PROGRAM ITAction
(*IMPORTANT !!! à modifier correctment selon les besoins*)
VAR CONSTANT
	//nombre total de dynamixel
	iNombreDynamixel 	: INT := 4;
	iNombreXL			: INT := 2;
	iNombreAX			: INT := 2;
	
	//définition de l'ID des dynamixels, tous les ID doivent se suivrent => ex: moteur_1 := 1,moteur_2 := 2, moteur_3 := 3, etc...
	//Si des moteurs AX-12A sont présents, leur ID doivent aller après celles des moteurs XL430 ou XL330 => ex: XL430_moteur_5 := 5, AX12A_moteur_1 := 6, etc...
	MoteurXL1 			: INT := 1; //exemple XL430
	MoteurXL2			: INT := 2;
	MoteurAX1 			: INT := 3; //exemple AX12A
	MoteurAX2			: INT := 4;
END_VAR	

VAR_INPUT
	//démarrage et arrêt du script python
	IbStartPyscript 	: BOOL;
	IbStopPyscript		: BOOL;

	//envoi de commande aux moteurs Dynamixel
	DXLIN 				: ARRAY [1..iNombreDynamixel] OF ST_Dynamixel_Control_Input;
END_VAR

VAR_OUTPUT
	QbPyScriptRunning 	: BOOL; //le script python est actif
	QiNombreDynamixel	: INT;
	//retour d'informations des moteurs Dynamixel
	DXLOUT 				: ARRAY [1..iNombreDynamixel] OF ST_Dynamixel_Control_Output;
END_VAR

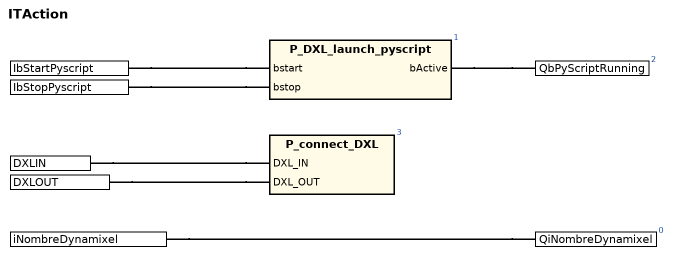
QiNombreDynamixel := iNombreDynamixel;
P_DXL_launch_pyscript(bstart := IbStartPyscript, bstop := IbStopPyscript);
QbPyScriptRunning := P_DXL_launch_pyscript.bActive;
P_connect_DXL(DXL_IN := DXLIN, DXL_OUT := DXLOUT);

END_PROGRAM

(* stored: Version 1.1.0.1, ProductVersion 3.1.4024.12
   POU ITAction: Id {d8c760c2-9596-4ce7-b98c-3b595645113e}, SpecialFunc None *)
